FUNCTION_BLOCK MONGO_WRAPPER
  {SET_ATTRIBUTE(OpcUa, SERVICE)}
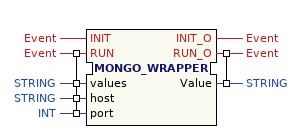
  EVENT_INPUT
    INIT;
    RUN WITH values, host, port; {SET_ATTRIBUTE(OpcUa, Method)}
  END_EVENT
  EVENT_OUTPUT
    INIT_O;
    RUN_O WITH Value;
  END_EVENT
  VAR_INPUT
    values : STRING; {SET_ATTRIBUTE(OpcUa, Variable.RUN)}
    host : STRING; {SET_ATTRIBUTE(OpcUa, Variable.RUN)}
    port : INT; {SET_ATTRIBUTE(OpcUa, Variable.RUN)}
  END_VAR
  VAR_OUTPUT
    Value : STRING; {SET_ATTRIBUTE(OpcUa, Variable.RUN)}
  END_VAR
END_FUNCTION_BLOCK
